# EPICS substitutions: iocStats/iocAdmin/Db/iocAdminScanMon.substitutions
#==============================================================================
#
# Abs:  IOC Administration Records for SCAN Monitoring
#
# Name: iocAdminScanMon.substitutions
#
#==============================================================================
#
file iocScanMon.template
{
#                                         0 = relative
#                                         1 = absolute    (%)         (%)
pattern { IOCNAME , SCANNAME   , SCAN        , MODE , MINOR_TOL , MAJOR_TOL }
	{ "$(IOC)"  , 01HZ       , "10 second" ,  1   ,   1.0     ,  10.0     }
	{ "$(IOC)"  , 02HZ       , "5 second"  ,  1   ,   1.0     ,  10.0     }
	{ "$(IOC)"  , 05HZ       , "2 second"  ,  1   ,   2.0     ,  10.0     }
	{ "$(IOC)"  , 1HZ        , "1 second"  ,  1   ,   2.0     ,  10.0     }
	{ "$(IOC)"  , 2HZ        , ".5 second" ,  1   ,   5.0     ,  10.0     }
	{ "$(IOC)"  , 5HZ        , ".2 second" ,  1   ,   5.0     ,  10.0     }
	{ "$(IOC)"  , 10HZ       , ".1 second" ,  1   ,   5.0     ,  10.0     }
}

file iocScanMonSum.template
{
pattern { IOCNAME , SCANNAME0 , SCANNAME1 , SCANNAME2 , SCANNAME3 , SCANNAME4 , SCANNAME5 , SCANNAME6 }
	{ "$(IOC)"  , 01HZ      , 02HZ      , 05HZ      , 1HZ       , 2HZ       , 5HZ       , 10HZ      }
}
